// Checks if a pointer is in a readable memory area (static/dynamic).
FUNCTION F_IsReadablePointer : BOOL // TRUE if the given pointer refers to a readable memory area.
VAR_INPUT
	// Pointer to check for readability.
	pValue : POINTER TO BYTE;
END_VAR
VAR
END_VAR

CASE F_GetAddressMemoryArea(pValue) OF 
	E_AddressMemoryArea.Static,
	E_AddressMemoryArea.Dynamic:
		F_IsReadablePointer := TRUE;
	END_CASE

END_FUNCTION

(* stored: Version 1.1.0.1
   POU F_IsReadablePointer: Id {64f8419c-84ee-0745-0049-c0fc706b418f}, SpecialFunc None *)
